{attribute addProperty BoxType "EL2262-0000-0001"}
{attribute addProperty Id "Output1AT %Q*BOOL81"}
{attribute addProperty CRC "1129441452"}
{attribute addProperty SizeInBites "8"}
{attribute addProperty SizeInBytes "1"}
TYPE Sample_4351E8AC :
STRUCT
	{attribute addProperty Name "Output1"}
	Output1 AT %Q* : BOOL;
END_STRUCT
END_TYPE

(* stored: Version 1.2.0.0, ProductVersion 3.1.4024.9
   DUT Sample_4351E8AC: Id {667b51db-9958-412b-8646-cccd93bffc53} *)
